TYPE st_yellow_visibility :
STRUCT
	main				:BOOL;
	recipe				:BOOL;
	graph				:BOOL;
	maintenance			:BOOL;
	io					:BOOL;
	auto_mode			:BOOL;
	debug_mode			:BOOL;
END_STRUCT
END_TYPE

(* stored: Version 1.1.0.1, ProductVersion 3.1.4020.12
   DUT st_yellow_visibility: Id {3ab271a0-2c98-44d2-978b-b8c6a3fbcca6} *)
